// TIA Portal V17 export
// export: Created 2024-08-09T12:50:43.9381424Z, ExportSetting WithDefaults, DisplayName Totally Integrated Automation Portal, DisplayVersion V17 Update 7, DisplayName TIA Portal Openness, DisplayVersion V17 Update 7, DisplayName TIA Portal Version Control Interface, DisplayVersion V17, DisplayName STEP 7 Professional, DisplayVersion V17 Update 7, DisplayName STEP 7 Safety, DisplayVersion V17 Update 6, DisplayName WinCC Professional, DisplayVersion V17 Update 7
DATA_BLOCK "DB_BIBLIOTHEQUE"   // DB3
{ S7_Optimized_Access := 'TRUE' }
VERSION : 0.1
// stored: AutoNumber true, DBAccessibleFromOPCUA true, DBAccessibleFromWebserver true, IsOnlyStoredInLoadMemory false, IsRetainMemResEnabled false, IsWriteProtectedInAS false, MemoryReserve 100
   VAR RETAIN
      Mobile : Array[0.."Nbr_Max_Mobiles"] of "S_Mobile";
      Lots_Taches { S7_SetPoint := 'True'} : Array[0.."Nbr_Max_Tache"] of "S_Lots_Tache";
      Zones_Suivi { S7_SetPoint := 'True'} : Array[0.."Nbr_Max_Lots"] of "S_Zone_Suiv_Lot";
      Defaut { S7_SetPoint := 'True'} : Array[0.."Nbr_Max_Def"] of "S_Defaut";
      D_IO { S7_SetPoint := 'True'} : Array[0..2999] of "S_D_IO";
   END_VAR
BEGIN
END_DATA_BLOCK
